(* IEC 61131-3 sources: CodesysTest/export/UN00 - Sharp Bagger/EM01 - Bagger Head/CM08 - Barcode Verifier/FB_BaseBCV.pou/BadRead.prop, 1 file *)

(* ---- Get.pm.st ---- *)
(*#-#-#-#-#-#-#-#-#-#---Declaration---#-#-#-#-#-#-#-#-#-#-#-#-#*)

VAR
END_VAR
(*#-#-#-#-#-#-#-#-#-#---Implementation---#-#-#-#-#-#-#-#-#-#-#-#-#*)

BadRead :=  _badread;
